Fanuc KAREL source: BYTES_AHEAD.kl

PROGRAM T
%NOLOCKGROUP
VAR
 v0 : FILE
 v1 : INTEGER
 v2 : INTEGER
BEGIN
 BYTES_AHEAD(v0, v1, v2)
END T
